(* CODESYS project motores.project
   CustomField01_name: CustomField01
   CustomField08_name: CustomField08
   CustomField06_name: CustomField06
   Title: ATV_IMC_Template
   CustomField09_name: CustomField09
   CustomField07_name: CustomField07
   CustomField05_name: CustomField05
   CustomField02_name: CustomField02
   Description: This template can be used for a correct interface with the local drive. the MANDATORY_AT_EACH_CYCLE program must be called like it is done in this application.
   CustomField04_name: CustomField04
   CustomField10_name: CustomField10
   Version: 0.0.0.0
   Company: Schneider Electric
   CustomField03_name: CustomField03

Project tree, tasks and I/O mapping:
  MyController : TM241CE24R, Schneider Electric, order no. TM241CE24R, version 4.0.2.9
    application Application
      task MAST (cyclic, interval 20 ms, priority 15, watchdog 100 ms x 1) calls nothing
      function HiddenPOU [ST]
      global variables GVL
      function block activacionmotor [LD]
      program motores [LD]
    DI : Digital Inputs, Schneider Electric, version 4.0.2.9
        input  iwDI_IW0 : WORD  // IW0
        input  ibDI_IB1 : BYTE  // IB1
    DQ : Digital Outputs, Schneider Electric, version 4.0.2.9
        output qwDQ_QW0 : WORD  // QW0
        output qbDQ_QB1 : BYTE  // QB1
    Counters : Counters, Schneider Electric, version 4.0.2.9
    Pulse_Generators : Pulse Generators, Schneider Electric, version 4.0.2.9
    Cartridge_1 : Cartridge, Schneider Electric, version 4.0.2.9
    IO_Bus : IO bus - TM3, Schneider Electric, version 4.0.2.9
    COM_Bus : COM bus, Schneider Electric, version 4.0.2.9
    Ethernet_1 : Ethernet Network, Schneider Electric, version 4.0.2.9
    Serial_Line_1 : Serial line, Schneider Electric, version 4.0.2.9
      SoMachine_Network_Manager : SoMachine-Network Manager, Schneider Electric, version 4.0.0.2
    Serial_Line_2 : Serial line, Schneider Electric, version 4.0.2.9
      Modbus_Manager : Modbus Manager, Schneider Electric, version 4.0.0.2
*)

// MyController/Application/GVL
VAR_GLOBAL
	etapa1: BOOL;
	etapa0: BOOL;
	TempMotor: TON;
END_VAR

// MyController/Application/HiddenPOU
FUNCTION HiddenPOU : BOOL

VAR_INPUT
	pHiddenFunc: POINTER TO WORD;
END_VAR
VAR
	pRead: POINTER TO BYTE;
	pWrite: POINTER TO BYTE;
END_VAR

pRead := pHiddenFunc + 400;
pWrite := pHiddenFunc + 4400;
HiddenPOU := TRUE;

END_FUNCTION

// MyController/Application/activacionmotor
FUNCTION_BLOCK activacionmotor
VAR_INPUT
	InInicio:BOOL;
	InParar:BOOL;
	InTempActivacion:INT;
	
END_VAR
VAR_OUTPUT
	OutLampara:BOOL;
	OutMotor:BOOL;
	OutFin:BOOL;
	
END_VAR
VAR
	BLINK_0: BLINK;
END_VAR
VAR // added by the converter: edge detectors and wires of the graphical bodies
    _w1, _w2, _w3 : BOOL;
END_VAR

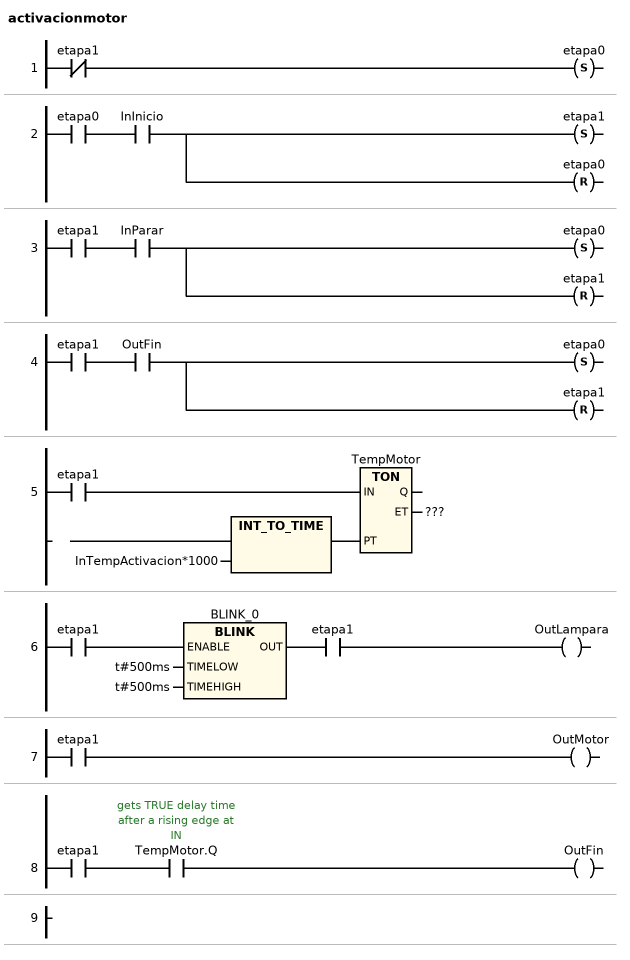
// NETWORK 1
etapa0 S= NOT etapa1;

// NETWORK 2
_w1 := etapa0 AND InInicio;
etapa1 S= _w1;
etapa0 R= _w1;

// NETWORK 3
_w2 := etapa1 AND InParar;
etapa0 S= _w2;
etapa1 R= _w2;

// NETWORK 4
_w3 := etapa1 AND OutFin;
etapa0 S= _w3;
etapa1 R= _w3;

// NETWORK 5
TempMotor(IN := etapa1, PT := INT_TO_TIME(InTempActivacion*1000)); // TON

// NETWORK 6
BLINK_0(ENABLE := etapa1, TIMELOW := t#500ms, TIMEHIGH := t#500ms); // BLINK
OutLampara := BLINK_0.OUT AND etapa1;

// NETWORK 7
OutMotor := etapa1;

// NETWORK 8
//   TempMotor.Q: gets TRUE delay time after a rising edge at IN
OutFin := etapa1 AND TempMotor.Q;

// NETWORK 9

END_FUNCTION_BLOCK

// MyController/Application/motores
PROGRAM motores
VAR
	Parpadeo1: BLINK;
	etapa0:BOOL;
	etapa1:BOOL;
	etapa2:BOOL;
	etapa3:BOOL;
	etapa4:BOOL;
	etapa5:BOOL;
	PEnviar:BOOL;
	MotorUser:INT;
	FinProceso:BOOL;
	TiempoActUser:INT;
	ActivMotor1: FB_ActivacionMotorTemp;
	ActivMotor2: FB_ActivacionMotorTemp;
	ActivMotor3: FB_ActivacionMotorTemp;
END_VAR
VAR_GLOBAL
	PMarcha:BOOL;
	LamparaOn:BOOL;
	PParo:BOOL;
	LamparaMotor1:BOOL;				
	Motor1:BOOL;
	LamparaMotor2:BOOL;
	Motor2:BOOL;
	LamparaMotor3:BOOL;
	Motor3:BOOL;
END_VAR
VAR // added by the converter: edge detectors and wires of the graphical bodies
    _w1, _w2, _w3, _w4, _w5, _w6, _w7, _w8 : BOOL;
END_VAR

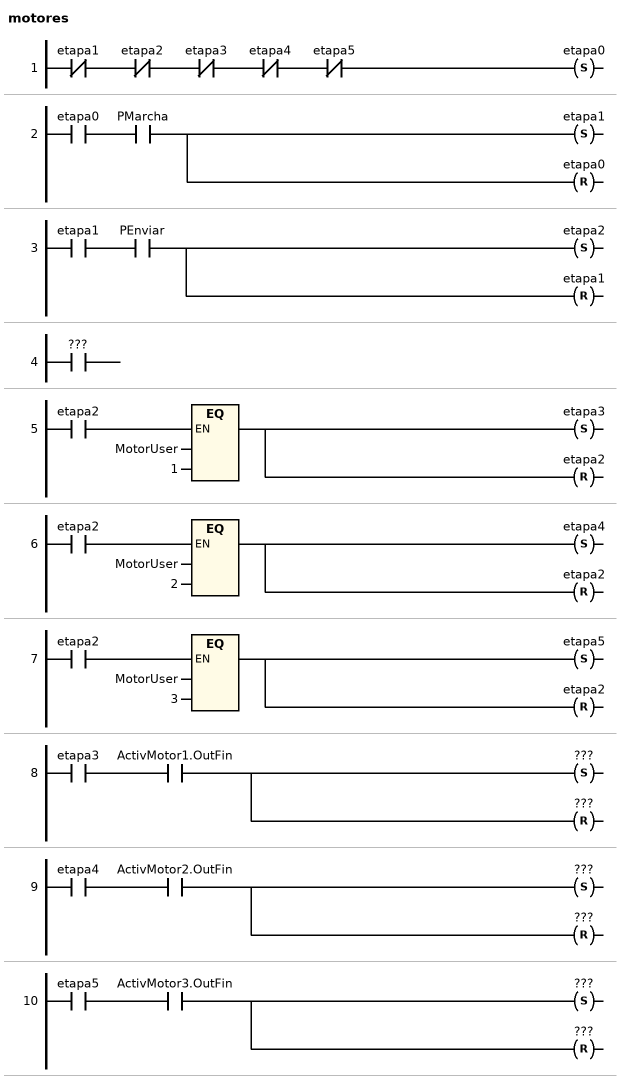
// NETWORK 1
etapa0 S= NOT etapa1 AND NOT etapa2 AND NOT etapa3 AND NOT etapa4 AND NOT etapa5;

// NETWORK 2
_w1 := etapa0 AND PMarcha;
etapa1 S= _w1;
etapa0 R= _w1;

// NETWORK 3
_w2 := etapa1 AND PEnviar;
etapa2 S= _w2;
etapa1 R= _w2;

// NETWORK 4

// NETWORK 5
_w3 := etapa2 AND MotorUser = 1;
etapa3 S= _w3;
etapa2 R= _w3;

// NETWORK 6
_w4 := etapa2 AND MotorUser = 2;
etapa4 S= _w4;
etapa2 R= _w4;

// NETWORK 7
_w5 := etapa2 AND MotorUser = 3;
etapa5 S= _w5;
etapa2 R= _w5;

// NETWORK 8
_w6 := etapa3 AND ActivMotor1.OutFin;
??? S= _w6;
??? R= _w6;

// NETWORK 9
_w7 := etapa4 AND ActivMotor2.OutFin;
??? S= _w7;
??? R= _w7;

// NETWORK 10
_w8 := etapa5 AND ActivMotor3.OutFin;
??? S= _w8;
??? R= _w8;

END_PROGRAM
